FUNCTION_BLOCK SS3_ps_Flipper (* Composite FB wrapping other FBs *)
  (* Standard: 61499-2 *)
  (* Version 1.0, 2025-08-24, PS_Transformer_for_Unknown *)
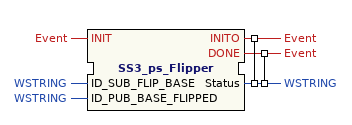
  EVENT_INPUT
    INIT; (* Initialization Request *)
  END_EVENT
  EVENT_OUTPUT
    INITO WITH Status; (* Initialization Confirm *)
    DONE WITH Status; (* Execution Confirmation *)
  END_EVENT
  VAR_INPUT
    ID_SUB_FLIP_BASE : WSTRING;
    ID_PUB_BASE_FLIPPED : WSTRING;
  END_VAR
  VAR_OUTPUT
    Status : WSTRING; (* Output event qualifier *)
  END_VAR
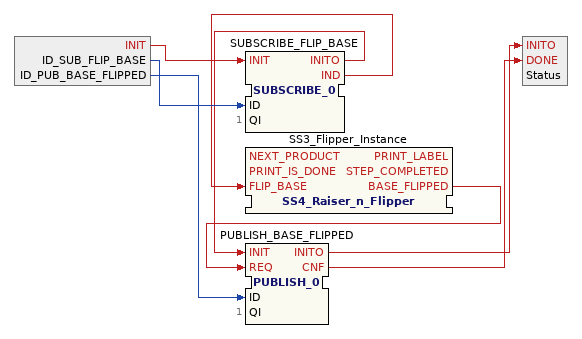
  FBS
    SS3_Flipper_Instance : SS4_Raiser_n_Flipper;
    SUBSCRIBE_FLIP_BASE : SUBSCRIBE_0(QI := 1);
    PUBLISH_BASE_FLIPPED : PUBLISH_0(QI := 1);
  END_FBS
  EVENT_CONNECTIONS
    INIT TO SUBSCRIBE_FLIP_BASE.INIT;
    SUBSCRIBE_FLIP_BASE.INITO TO PUBLISH_BASE_FLIPPED.INIT;
    PUBLISH_BASE_FLIPPED.INITO TO INITO;
    SUBSCRIBE_FLIP_BASE.IND TO SS3_Flipper_Instance.FLIP_BASE;
    SS3_Flipper_Instance.BASE_FLIPPED TO PUBLISH_BASE_FLIPPED.REQ;
    PUBLISH_BASE_FLIPPED.CNF TO DONE;
  END_CONNECTIONS
  DATA_CONNECTIONS
    ID_SUB_FLIP_BASE TO SUBSCRIBE_FLIP_BASE.ID;
    ID_PUB_BASE_FLIPPED TO PUBLISH_BASE_FLIPPED.ID;
  END_CONNECTIONS
END_FUNCTION_BLOCK
